FUNCTION TryConvert_SINT_TO_BOOL : BOOL
VAR_INPUT
	in : SINT;
	out : REFERENCE TO BOOL;
END_VAR

out := SINT_TO_BOOL(in);
TryConvert_SINT_TO_BOOL := TRUE;

END_FUNCTION

(* stored: Version 1.1.0.1, ProductVersion 3.1.4024.12
   POU TryConvert_SINT_TO_BOOL: Id {cbbd89b9-3b22-4b51-a41c-7e26a87f268e}, SpecialFunc None *)
